StartStopCommand_213();
StartStopStatus_213();
Alarm_213();
MalfunctionCode_213();




RoomTemp_213();
TempAdjust_213();
FilterSign_213();
FilterSignReset_213();
RemoteControlStart_213();

RemoteControlTempAdjust_213();












StartStopCommand_224();
StartStopStatus_224();
Alarm_224();
MalfunctionCode_224();




RoomTemp_224();
TempAdjust_224();
FilterSign_224();
FilterSignReset_224();
RemoteControlStart_224();

RemoteControlTempAdjust_224();












StartStopCommand_225();
StartStopStatus_225();
Alarm_225();
MalfunctionCode_225();




RoomTemp_225();
TempAdjust_225();
FilterSign_225();
FilterSignReset_225();
RemoteControlStart_225();

RemoteControlTempAdjust_225();












StartStopCommand_226();
StartStopStatus_226();
Alarm_226();
MalfunctionCode_226();




RoomTemp_226();
TempAdjust_226();
FilterSign_226();
FilterSignReset_226();
RemoteControlStart_226();

RemoteControlTempAdjust_226();












StartStopCommand_227();
StartStopStatus_227();
Alarm_227();
MalfunctionCode_227();




RoomTemp_227();
TempAdjust_227();
FilterSign_227();
FilterSignReset_227();
RemoteControlStart_227();

RemoteControlTempAdjust_227();












StartStopCommand_241();
StartStopStatus_241();
Alarm_241();
MalfunctionCode_241();




RoomTemp_241();
TempAdjust_241();
FilterSign_241();
FilterSignReset_241();
RemoteControlStart_241();

RemoteControlTempAdjust_241();












StartStopCommand_243();
StartStopStatus_243();
Alarm_243();
MalfunctionCode_243();




RoomTemp_243();
TempAdjust_243();
FilterSign_243();
FilterSignReset_243();
RemoteControlStart_243();

RemoteControlTempAdjust_243();












CL_Rejection_000();
SystemForcedOff_000();
CL_Rejection_064();
SystemForcedOff_064();
CL_Rejection_128();
SystemForcedOff_128();
CL_Rejection_192();
SystemForcedOff_192();

END_FUNCTION_BLOCK

(* stored: Version 1.1.0.1, ProductVersion 3.1.4024.14
   POU FB_BACnet_DAIKIN_MasterStation_III_No_8: Id {2cdd84e9-cbd7-4cbb-a552-a66c20b14db1}, SpecialFunc None *)
